FUNCTION_BLOCK DINT2DINT
  {SET_ATTRIBUTE(OpcUa, SERVICE)}
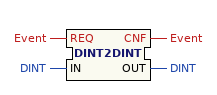
  EVENT_INPUT
    REQ;
  END_EVENT
  EVENT_OUTPUT
    CNF;
  END_EVENT
  VAR_INPUT
    IN : DINT;
  END_VAR
  VAR_OUTPUT
    OUT : DINT;
  END_VAR
END_FUNCTION_BLOCK
